(* CODESYS project amko_system.library
   Author: Chris van Kooij
   Placeholder: System_Library
   Title: System_Library
   Version: 0.0.0.3
   Description: system and module base functions
   Company: AMKO-Engineering

Project tree, tasks and I/O mapping:
  libraries: Device_Library, * (AMKO-Engineering); Tc2_Standard, * (Beckhoff Automation GmbH); Tc2_System, * (Beckhoff Automation GmbH); Tc2_Utilities, * (Beckhoff Automation GmbH); Utilities_Library, * (AMKO-Engineering)
  FaultHandler/
    function block Fb_SystemFaultHandler [ST]: CheckForModuleFaults, ExecMessageCompare, ExecScreenControl, ExecSetFaultBit, ExecWriteToLog
  GVLs/
    global variables GVL_Main
  ModuleBase/
    Base/
      function block Fb_ModuleBase [ST]: CmdAutomatic, CmdEstop, CmdHold, CmdHome, CmdInit, CmdPowerOff, CallComponents, CheckCollision, ExecAutomatic, ExecHold, ExecHome, ExecInit, ExecManual, ExecPowerOff, ExecReset, ExecSafeStop, ExecFaultHandling, ExecMainBaseFunctions
    DataTypes/
      data type Udt_ModuleBase
  SystemBase/
    DataTypes/
      data type E_StateSystem
      data type Udt_ModuleId
    program SystemBase [ST]: CallModules, ExecAutomatic, ExecHoming, ExecPowerOff, ExecSafeHold, ExecSafeReset, ExecSafeStop, Init, CallSystemFunctions, CheckSystemOK, ExecSystemRun, CmdAddModule
*)

// ModuleBase/DataTypes/Udt_ModuleBase
TYPE Udt_ModuleBase :
STRUCT
	sModuleName 		: STRING := 'NA' 		; // Module name
	bModuleActive		: 	BOOL := FALSE 		; // Module is active in the system (will be ignored by system if false) 	
	// safety Inputs
	bEstopOk			:	BOOL ; // When estop is not ok, complete machine is shut down and reinitialization is required.
	bModuleSafetyOk		: 	BOOL ; // Module safety systems are ok and safe 
	bAirPressureOk		: 	BOOL ; // system safety condition monitorring air pressure ok
	bPowerSupplyOk		: 	BOOL ; // System power supply is ok
	// main system Inputs
	bCmdStart			: 	BOOL	:= FALSE ; // System start command 
	bCmdReset 			: 	BOOL	:= FALSE ; // reset all faults 
	bCmdPowerOff		:	BOOL	:= FALSE ; // power off module 
	bCmdStartManual 	: 	BOOL 	:= FALSE ; // Start up in manual mode
 	// Com to main system
	fbFaultHandler		: 	Fb_FaultHandler 		; // Fault handler 
	sStateIndicator		: 	STRING := ''			; // Operator message, indication of current step or function 

	// Fault indications
	bMissingCond	: BOOL := FALSE ; // Module missing condition active
	bFatalFault		: BOOL := FALSE ; // Module fatal fault is active
	bCycleFault		: BOOL := FALSE ; // Module cycle fault is active

	// State indication
	bIsSafe			: BOOL := FALSE ; // Module is safe and locked until safety is ok
	bNoreference	: BOOL := FALSE ; // Module Startup Undefined initialization required

	bInitializing	: BOOL := FALSE ; // Module startup initializing
	binitialized	: BOOL := FALSE ; // Module startup initialized waiting for startup command

	bIdle 			: BOOL := FALSE ; // Module startup Idle no commands active

	bEnabling 		: BOOL := FALSE ; // Module Startup enabeling 
	bEnabled 		: BOOL := FALSE ; // Module Startup Enabled
	
	bHoming			: BOOL := FALSE ; // Module startup homing back to base position and recalibrate
	bHomed 			: BOOL := FALSE ; // Module startup homed waiting for further further commands

	bHolding 		: BOOL := FALSE ; // Module Module Hold motion command executing
	bHeld	 		: BOOL := FALSE ; // Module Hold Motion is held until command is released	
	
	bResetting 		: BOOL := FALSE ; // Module Reset resetting error status
	bResetDone 		: BOOL := FALSE ; // Module reset is done   

	bManual 		: BOOL := FALSE ; // Module Work status Module in Manual 
	bAutomatic 		: BOOL := FALSE ; // Module Work status Module in Automatic mode
	
	bPoweringOff	: BOOL := FALSE ; // Module is powering off
	bPowerdOff		: BOOL := FALSE ; // Module has powerd off 	
	
	// manual functions 
	bDevicesAddedtoManual	: BOOL := FALSE ;
	bParametersAdded		: BOOL := FALSE ;
	// Persistent data
	bCmdWritePersistent  : BOOL := false ; // write persistent data to memory
END_STRUCT
END_TYPE

// SystemBase/DataTypes/E_StateSystem
{attribute 'qualified_only'}
{attribute 'strict'}
{attribute 'to_string'}
TYPE E_StateSystem :
(
	NoReference		, 	// system has not been initialized
	Initialize		, 	// System is initializing
	LoadParameters	, 	// System is loading parameters from/to file
	Enable			, 	// System is enabling 
	Home			, 	// system is hominig 
	Reset			, 	// System is resetting
	Idle			, 	// system is waiting for commands
	Manual			, 	// System is in manual mode
	Automatic		, 	// system is in automatic mode 
	PowerOff		// system is powering off
)INT;
END_TYPE

// SystemBase/DataTypes/Udt_ModuleId
TYPE Udt_ModuleId :
STRUCT
	nNumber		: UDINT ; // Module identification number used for sorting order
	sName		: STRING; // Module name
	pFunction	: POINTER TO Fb_ModuleBase ;
END_STRUCT
END_TYPE

// GVLs/GVL_Main

{attribute 'qualified_only'} // Main system variables and state indicators
VAR_GLOBAL CONSTANT
	cnMaxNUMBEROFMODULES 	: UDINT := 10 		; // "maximum" number of modules in the system
	CtAIRPRESSUREDELAY	: TIME 	:= T#500MS	; // Timout before air fault becomes active
	cbUPSPRESENT		: BOOL	:= FALSE 	; // Enable automatic shutdown when power is interupted
END_VAR
VAR_GLOBAL PERSISTENT
	nTotalUnitsProduced		: UDINT ; // Units produced 
END_VAR

// FaultHandler/Fb_SystemFaultHandler
FUNCTION_BLOCK INTERNAL Fb_SystemFaultHandler
VAR_INPUT
	nNumberOfModules	: UDINT ; // Number of modules connected to the system fault handler
END_VAR
VAR_IN_OUT
	arpModules			: ARRAY [0..gvl_main.cnMaxNUMBEROFMODULES] OF Udt_ModuleId ;
END_VAR
VAR_OUTPUT
	// Fault types 
	bSystemFF			: BOOL 	:= FALSE	; // System fatal fault is active
	bSystemCF			: BOOL 	:= FALSE	; // System Cycle fault is active
	bSystemMC 			: BOOL 	:= FALSE	; // a missing condition is active only 
END_VAR
VAR
	// Message variables
	bResetFaults		: REFERENCE TO BOOL 	:= GVL_Message.bResetFaults		; // Reset system faults 
	bCmdSnoozeMessage	: REFERENCE TO BOOL  	:= GVL_Message.bCmdSnoozeMessage; // Snooze message display
	arActiveFaults 		: REFERENCE TO ARRAY [0..Param_Messages.nMAX_MESSAGES_SHOWN] OF UDT_Fault := GVL_Message.arActiveFaults ; // Active faults overview for showing in HMI
	arOldFaults 		: ARRAY [0..Param_Messages.nMAX_MESSAGES_SHOWN] OF UDT_Fault ; // Old faults overview for comparing to active
	arWriteToLog		: ARRAY [0..Param_Messages.nMAX_MESSAGES_SHOWN] OF UDT_Fault ; // Fault array for writing to log file 
	// Message logging
	dToday				: DATE 	; 
	nWriteStep			: UDINT := 0 ;
	bWriteError			: BOOL 	; // write to file error occured
	nWriteErroId		: UDINT ; // write error id
	// Write variables
	sActFileName		: STRING;
	hFile				: UINT	:= 0;(* File handle of the source file *)
	sMessageString		: ARRAY [0..Param_Messages.nMESSAGE_COLUMNS] OF STRING (GVL_Parameters.MAX_CSV_FIELD_LENGTH); (* temporary parameter buffer to string*)
	sCSVLine			: T_MaxString := '';(* Single CSV text line (row, record), we are using string as record buffer (your are able to see created fields) *)
	sCSVField			: T_MaxString := '';(* Single CSV field value (column, record field) *)
END_VAR
VAR // functions 
	tofSnoozeMessages	: TOF ; // timer function for message snoozing
	// Log to file functions
	fbFileOpen		: FB_FileOpen	;(* Opens file *)
	fbFileClose		: FB_FileClose	;(* Closes file *)
	fbFileGets		: FB_FileGets	;(* Reads one record (line) *)
	fbFilePuts		: FB_FilePuts	;(* Writes one record (line) *)
	fbReader		: FB_CSVMemBufferReader;(* Helper function block used to parse CSV data bytes (single record line) *)
	fbWriter		: FB_CSVMemBufferWriter;(* Helper function block used to create CSV data bytes (single record line) *)
END_VAR 
VAR CONSTANT
	stEmptyMessageUdt : UDT_Fault := (	Active 			:= FALSE,
									FaultType 		:= E_FaultTypes.NA,
									MessageNumber	:= 0,
									LocationNumber	:= 0,
									Discription 	:= '',
									LocationName	:= '',
									ComponentType	:= E_ComponentTypes.NA,
									StartTime		:= DT#2020-1-1-00:00:00,
									EndTime			:= DT#2020-1-1-00:00:00,
									FullFaultId		:= '0'	)  ;
END_VAR

// Check modules for active messages 
CheckForModuleFaults();
// set system fault bits 
ExecSetFaultBit(); 
// Message Screen controller 
ExecScreenControl();
// Log faults when they are reset
ExecMessageCompare();
// Logfile writer 
ExecWriteToLog();

METHOD PRIVATE CheckForModuleFaults : BOOL // check all modules for faults and copy them to the main fault array
VAR
	// functional variables
	i 					: UDINT ;
	j 					: UDINT ;
	// temporary fault storage
	arTempFaults	: ARRAY [0..Param_Messages.nMAX_MESSAGES_SHOWN] OF UDT_Fault ; // internal fault array
	p				: UDINT	;
END_VAR
// Go over modules to check for fault messages 
FOR i := 0 TO nNumberOfModules DO 
	// Check for active messages
	FOR j := 0 TO Param_Messages.nMAX_MESSAGES_SHOWN DO 
		IF arpModules[i].pFunction^.fbFaultHandler.arActiveFaults[j].FaultType <> E_FaultTypes.NA THEN 
			arTempFaults[p]:= arpModules[i].pFunction^.fbFaultHandler.arActiveFaults[j] ;
			p := MAX( p + 1, Param_Messages.nMAX_MESSAGES_SHOWN)  ;
		ELSE
			EXIT ;
		END_IF
	END_FOR
END_FOR

arOldFaults		:= arActiveFaults 	;
arActiveFaults	:= arTempFaults 	;
END_METHOD

METHOD PRIVATE ExecMessageCompare : BOOL
VAR
	// functional variables
	i 			: UDINT ;
	j 			: UDINT ;
	bFaultFound : BOOL ;
	p			: UDINT;
END_VAR
// Check if any changes occured in the active faults
FOR i := 0 TO Param_Messages.nMAX_MESSAGES_SHOWN DO
	// break loop if fault is empty
	IF  arOldFaults[i].FaultType = E_FaultTypes.NA THEN  
		EXIT;
	ELSE
		// check if the fault is still active
		bFaultFound := TRUE; 
		FOR j := 0 TO Utilities_Library.Param_Messages.nMAX_MESSAGES_SHOWN DO
			bFaultFound := arOldFaults[i].FullFaultId = arActiveFaults[j].FullFaultId AND bFaultFound ;
		END_FOR
		// if the fault is not faund then wrtie it to the logging array for loging
		IF NOT bFaultFound THEN 
			arWriteToLog[p] := arOldFaults[i] ;
			p := p + 1 ; 
		END_IF
	END_IF
END_FOR
END_METHOD

METHOD PRIVATE ExecScreenControl : BOOL // Control message screen 
VAR_INPUT
END_VAR
tofSnoozeMessages(IN := bCmdSnoozeMessage, PT := GVL_Message.tMESSAGESNOOZEDURATION);

// Set screen control 
IF bSystemCF OR bSystemFF THEN 
	GVL_Message.bHideFaults := FALSE ;
ELSIF bSystemMC AND NOT tofSnoozeMessages.Q THEN 
	GVL_Message.bHideFaults := FALSE ;
ELSE
	GVL_Message.bHideFaults := TRUE ;
END_IF
END_METHOD

METHOD PRIVATE ExecSetFaultBit : BOOL
VAR
	// functional variables
	i 			: UDINT ;
END_VAR
bSystemFF	:= FALSE ;
bSystemCF	:= FALSE ;
bSystemMC	:= FALSE ;

FOR i := 0 TO Param_Messages.nMAX_MESSAGES_SHOWN DO
	bSystemFF	:= arActiveFaults[i].FaultType = E_FaultTypes.FF OR bSystemFF;
	bSystemCF	:= arActiveFaults[i].FaultType = E_FaultTypes.CF OR bSystemCF;
	bSystemMC	:= arActiveFaults[i].FaultType = E_FaultTypes.MC OR bSystemMC;
END_FOR
END_METHOD

METHOD PRIVATE ExecWriteToLog : BOOL
VAR 
	i : UDINT ; 
	p : UDINT ; // Fault array pointer
END_VAR
dToday := DT_TO_DATE(Sys_Variables.SystemTime);
// create file name with Current date 
sActFileName 	:= CONCAT(STR1 := Param_Messages.sLOGFILE_PATH	, STR2 := Param_Messages.sLOGFILE_NAME	);
sActFileName 	:= CONCAT(STR1 := sActFileName					, STR2 := DATE_TO_STRING(dToday)		);
sActFileName 	:= CONCAT(STR1 := sActFileName					, STR2 := '.csv'						);

// ===== Start file write =====
CASE nWriteStep OF
	0:	(* Wait until log array is filled *)
		IF arWriteToLog[0].FaultType <> E_FaultTypes.NA THEN 
			hFile				:= 0;
			nWriteStep 			:= 1;
		ELSE 
			RETURN ;
		END_IF
	1:	(* Open source file *)
		fbFileOpen(  bExecute := FALSE  );
		fbFileOpen( sNetId := GVL_Parameters.sNetId, sPathName := sActFileName , nMode := FOPEN_MODEAPPEND OR FOPEN_MODETEXT,(* Open file in TEXT mode! *)
					ePath := PATH_GENERIC, bExecute := TRUE );
		nWriteStep := nWriteStep + 1 ;
	2:(* Wait until open not busy *)
		fbFileOpen( bExecute := FALSE, bError => bWriteError, nErrID => nWriteErroId, hFile => hFile );
		IF NOT fbFileOpen.bBusy THEN
			IF NOT fbFileOpen.bError THEN
				nWriteStep := nWriteStep + 1 ;
			ELSE(* Error: file not found? *)
				nWriteStep := 100;
			END_IF
		END_IF
	3: (* Check if faultrecord is active if so skip record *)
		nWriteStep := nWriteStep + 1 ;
	4:(* Convert one PLC record to CSV format *)
		sCSVLine := '';
		fbWriter.eCmd := eEnumCmd_First;(* Write first field value *)
		// write message data to string
		sMessageString[0] 	:= TO_STRING(arWriteToLog[p].FaultType				);
		sMessageString[1]	:= DT_TO_STRING(arWriteToLog[p].StartTime			);
		sMessageString[2]	:= DT_TO_STRING(Sys_Variables.SystemTime			);
		sMessageString[3]	:= UDINT_TO_STRING(arWriteToLog[p].MessageNumber	);
		sMessageString[4]	:= UDINT_TO_STRING(arWriteToLog[p].LocationNumber	); 
		sMessageString[5]	:= arWriteToLog[p].Discription						;
		sMessageString[6]	:= arWriteToLog[p].LocationName						;
		sMessageString[7]	:= TO_STRING(arWriteToLog[p].ComponentType			);
		// write data to .csv buffer 
		FOR i := 0 TO Param_Messages.nMESSAGE_COLUMNS BY 1 DO
			sCSVField := STRING_TO_CSVFIELD(in :=  sMessageString[i], FALSE );
			(* Add new field to the record buffer *)
			fbWriter( 	pBuffer := ADR( sCSVLine ), cbBuffer := SIZEOF( sCSVLine ) - 1, putValue := sCSVField, pValue := 0, cbValue := 0,
						bCRLF := ( i = Param_Messages.nMESSAGE_COLUMNS ) );(* bCRLF == TRUE => Write CRLF after the last field value *)
			IF fbWriter.bOk THEN
				fbWriter.eCmd := eEnumCmd_Next;
			ELSE
				nWriteStep := 100;
				RETURN;
			END_IF
		END_FOR(* FOR nColumn := 0... *)

		(* FB_FilePuts adds allready CR (carriage return) to the written line.
		We have to replace the $R$L characters with $L character to avoid double CR. *)
		IF RIGHT( sCSVLine, 2 ) = '$R$L' THEN
			sCSVLine := REPLACE( sCSVLine, '$L', 2, LEN( sCSVLine ) - 1 );
		END_IF
		nWriteStep := nWriteStep + 1 ;
	5:	(* Write single text line to file *)
		fbFilePuts( bExecute := FALSE );
		fbFilePuts( sNetId := GVL_Parameters.sNetId, hFile := hFile, sLine := sCSVLine, bExecute := TRUE );
		nWriteStep := nWriteStep + 1 ;
	6:(* Wait until write not busy *)
		fbFilePuts( bExecute := FALSE, bError => bWriteError, nErrID => nWriteErroId );
		IF NOT fbFilePuts.bBusy THEN
			IF NOT fbFilePuts.bError THEN
				nWriteStep := nWriteStep + 1 ;
			ELSE(* Error *)
				nWriteStep := 100;
			END_IF
		END_IF
	7: (* clear fault from array and go to next fault *)
		arWriteToLog[p]:= stEmptyMessageUdt;
		IF p < Param_Messages.nMAX_MESSAGES_SHOWN THEN 
			p := p +1 ;
		END_IF
		nWriteStep := nWriteStep +1 ;
	8: (* If fault is active then repeat previous step, else close file*)		
		IF  arWriteToLog[p].FaultType <> E_FaultTypes.NA THEN 
			nWriteStep := 3 ;
		ELSE
			nWriteStep := 10;
		END_IF
	10:	(* Close source file *)
		fbFileClose( bExecute := FALSE );
		fbFileClose( sNetId := GVL_Parameters.sNetId, hFile := hFile, bExecute := TRUE );
		nWriteStep := 11;
	11:(* Wait until close not busy *)
		fbFileClose( bExecute := FALSE, bError => bWriteError, nErrID => nWriteErroId );
		IF ( NOT fbFileClose.bBusy ) THEN
			hFile 		:= 0;
			nWriteStep 	:= 100;
		END_IF
	100: (* Error or ready nWriteStep => cleanup *)
		IF ( hFile <> 0 ) THEN
			nWriteStep	:= 10; (* Close the source file *)
		ELSE
			nWriteStep 	:= 0;	(* Ready *)
			ExecWriteToLog := TRUE ;
		END_IF
END_CASE
END_METHOD

END_FUNCTION_BLOCK

// ModuleBase/Base/Fb_ModuleBase
{attribute 'reflection'}
FUNCTION_BLOCK PUBLIC ABSTRACT Fb_ModuleBase
VAR_INPUT
	nModuleID			: 	UDINT 	:= 1 	; // module reference number used for fault, enable, reset, and safety functions (default := 1, 0 = main system)
	// main system Inputs
	bEnable				: 	BOOL	:= FALSE ; // (autolinked) module enable 	
	bCmdReset 			: 	BOOL	:= FALSE ; // (AutoLinked) reset all faults 
	bSysFatalFault		: 	BOOL 	:= FALSE ; // (AutoLinked) System fatal fault active
	bSysCycleFault		: 	BOOL 	:= FALSE ; // (AutoLinked) System fatal fault active 
	// Internal safety 
	bSafetyOK			: BOOL := FALSE ; // Module internal safety is ok
END_VAR
VAR_OUTPUT
	sName 				: STRING 	:= 'NA' 			; // Module name
	bAddedToSystem		: BOOL 		:= FALSE 			; // module has been added to the system
 	// Com to main system
	fbFaultHandler		: 	Fb_FaultHandler 		; // Fault handler 
	sStateIndicator		: 	STRING := ''			; // Operator message, indication of current step or function 

	// Fault indications
	bMissingCond	: BOOL := FALSE ; // Module missing condition active
	bFatalFault		: BOOL := FALSE ; // Module fatal fault is active
	bCycleFault		: BOOL := FALSE ; // Module cycle fault is active

	// State indication
	bIsSafe			: BOOL := FALSE ; // Module is safe and locked until safety is ok
	bNoreference	: BOOL := FALSE ; // Module Startup Undefined initialization required
	binitialized	: BOOL := FALSE ; // Module startup initialized waiting for startup command
	bHomed 			: BOOL := FALSE ; // Module startup homed waiting for further further commands

	bHolding 		: BOOL := FALSE ; // Module Module Hold motion command executing
	bHeld	 		: BOOL := FALSE ; // Module Hold Motion is held until command is released	
	
	bResetDone 		: BOOL := FALSE ; // Module reset is done   

	bManual 		: BOOL := FALSE ; // Module Work status Module in Manual
	bStartAuto		: BOOL := FALSE ; // Module start automatic cycle 
	bAutomatic 		: BOOL := FALSE ; // Module Work status Module in Automatic mode
	
	bPoweringOff	: BOOL := FALSE ; // Module is powering off
	bPowerdOff		: BOOL := FALSE ; // Module has powerd off 	

END_VAR
VAR 
	// manual functions 
	bParametersAdded		: BOOL := FALSE ;
	// Persistent data
	bCmdWritePersistent  : BOOL := false ; // write persistent data to memory
	// Module data
	stMessage				: UDT_Fault			; // Message data
	// Function path 
	{attribute 'instance-path'} 
    {attribute 'noinit'}
	sPath			: STRING	; // Path name of function (used for manual reference)
END_VAR


// Get device name from function
IF sName = 'NA' THEN 
	sName := F_FBNameFromPath(sPath := sPath);
END_IF

// Add module to system
IF NOT bAddedToSystem THEN
	bAddedToSystem S= SystemBase.CmdAddModule(refToModule := THIS^);
END_IF

// Execute functions
ExecMainBaseFunctions();

METHOD INTERNAL CmdAutomatic : BOOL
VAR_INPUT
END_VAR
bStartAuto 		:= TRUE ;

CmdAutomatic 	:= bAutomatic;
END_METHOD

METHOD INTERNAL CmdEstop : BOOL
VAR_INPUT
END_VAR
ExecSafeStop();
bHomed			:= FALSE ;
bAutomatic 		:= FALSE ;


CmdEstop := bIsSafe ;
END_METHOD

METHOD INTERNAL CmdHold : BOOL
VAR_INPUT
END_VAR
bAutomatic 	:= FALSE ;
ExecHold();


CmdHold := bHeld ;
END_METHOD

METHOD INTERNAL CmdHome : BOOL
VAR_INPUT
END_VAR
ExecHome();

CmdHome := bHomed;
END_METHOD

METHOD INTERNAL CmdInit : BOOL
VAR_INPUT
END_VAR
ExecInit();

CmdInit := binitialized;
END_METHOD

METHOD INTERNAL CmdPowerOff : BOOL
VAR_INPUT
END_VAR
ExecPowerOff();
bAutomatic := FALSE ;

CmdPowerOff := bPowerdOff;
END_METHOD

METHOD PROTECTED ABSTRACT CallComponents : BOOL
VAR_INPUT
END_VAR
END_METHOD

METHOD PUBLIC ABSTRACT CheckCollision : BOOL // Checks device commands for positble collisions  and block if necesarry
VAR_INPUT
END_VAR
END_METHOD

METHOD PROTECTED ABSTRACT ExecAutomatic : BOOL
VAR_INPUT
END_VAR
END_METHOD

METHOD PROTECTED ABSTRACT ExecHold : BOOL
VAR_INPUT
END_VAR
END_METHOD

METHOD PROTECTED ABSTRACT ExecHome : BOOL
VAR_INPUT
END_VAR
END_METHOD

METHOD PROTECTED ABSTRACT ExecInit : BOOL
VAR_INPUT
END_VAR
END_METHOD

METHOD PROTECTED ExecManual : BOOL
VAR_INPUT
END_VAR
END_METHOD

METHOD PROTECTED ABSTRACT ExecPowerOff : BOOL
VAR_INPUT
END_VAR
END_METHOD

METHOD PROTECTED ABSTRACT ExecReset : BOOL
VAR_INPUT
END_VAR
END_METHOD

METHOD PROTECTED ABSTRACT ExecSafeStop : BOOL
VAR_INPUT
END_VAR
END_METHOD

METHOD ExecFaultHandling : BOOL
VAR_INPUT
END_VAR
// Call reset functions
IF bCmdReset THEN 
	fbFaultHandler.bReset := TRUE ;
	ExecReset();
END_IF

// Call message function
fbFaultHandler(bReset := bCmdReset);

bFatalFault := fbFaultHandler.bActFF ;
bCycleFault := fbFaultHandler.bActCF ;

IF bFatalFault THEN
	ExecSafeStop()	;
	binitialized	:= FALSE; 
	bHomed			:= FALSE;
ELSIF bCycleFault THEN
	bHeld			S= ExecHold();
	bHolding 		:= NOT bHeld ;
END_IF

// Reset safe state when enable is active
bIsSafe R= bEnable ;

// Prevent automatic start when fault is active
bStartAuto R= bCmdReset OR bFatalFault OR bCycleFault ;
END_METHOD

METHOD INTERNAL ExecMainBaseFunctions : BOOL
VAR_INPUT
END_VAR
// Check for anny Internal collisions
CheckCollision();

// Call components 
CallComponents();

// Call fault handling function 
ExecFaultHandling();

// Run automatic function 
IF bStartAuto THEN 
	bAutomatic := ExecAutomatic();
	bStartAuto :=FALSE ;
ELSE
	bAutomatic := FALSE ;
END_IF

// Persistent data 
IF bCmdWritePersistent THEN 
	bCmdWritePersistent R= DataManager.FbPersistentManager.Write();
END_IF
END_METHOD

END_FUNCTION_BLOCK

// SystemBase/SystemBase
{attribute 'reflection'}
PROGRAM SystemBase // system base program, from here all modules are controlled and the system functions are called.
VAR_IN_OUT
	// HMI Screens 
	nHMIShownscreen	: INT ; // show visualization screen (0 = default home screen, 1 = automatic screen, 2 =< configurable) 
END_VAR
VAR
	// Fault indications
	bMissingCond	: BOOL := FALSE ; // Module missing condition active
	bFatalFault		: BOOL := FALSE ; // Module fatal fault is active
	bCycleFault		: BOOL := FALSE ; // Module cycle fault is active

	// State indication
	bIsSafe			: BOOL := FALSE ; // Module is safe and locked until safety is ok
	bNoreference	: BOOL := FALSE ; // Module Startup Undefined initialization required

	bInitializing	: BOOL := FALSE ; // Module startup initializing
	binitialized	: BOOL := FALSE ; // Module startup initialized waiting for startup command

	bIdle 			: BOOL := FALSE ; // Module startup Idle no commands active

	bEnabling 		: BOOL := FALSE ; // Module Startup enabeling 
	bEnabled 		: BOOL := FALSE ; // Module Startup Enabled
	
	bHoming			: BOOL := FALSE ; // Module startup homing back to base position and recalibrate
	bHomed 			: BOOL := FALSE ; // Module startup homed waiting for further further commands

	bHolding 		: BOOL := FALSE ; // Module Module Hold motion command executing
	bHeld	 		: BOOL := FALSE ; // Module Hold Motion is held until command is released	
	
	bResetting 		: BOOL := FALSE ; // Module Reset resetting error status
	bResetDone 		: BOOL := FALSE ; // Module reset is done   

	bManual 		: BOOL := FALSE ; // Module Work status Module in Manual 
	
	bStartAuto		: BOOL := FALSE ; // Start automatic mode
	bAutomatic 		: BOOL := FALSE ; // Module Work status Module in Automatic mode
	
	bPoweringOff	: BOOL := FALSE ; // Module is powering off
	bPowerdOff		: BOOL := FALSE ; // Module has powerd off 	

END_VAR
VAR
	// System inputs 
	ibEstopOk 			AT%I*	: BOOL  ; // system emergency stop ok
	ibSystemSafetyOK	AT%I*	: BOOL  ; // System is safe 
	ibPowerSupplyOk	 	AT%I*	: BOOL  ; // System Power supply is ok 
	fbAirpressureOk 			: Fb_DevDigitalInputFunctions  	; // system airpressure is ok
	fbCmdResetSafety		 	: FB_DevPushbuttonLight 		; // System reset
	
	// System safety valve
	fbValveMainAirSupply		: FB_DevValve ; // Main air supply valve 
	
	// system Commands 
	fbCmdStartSystem		 	: FB_DevPushbuttonLight  		; // (re)start system input from button
	fbCmdStartManual			: FB_DevHMIButton 				; // Start system in manual mode 
	fbCmdPowerOff				: FB_DevHMIButton 				; // Power off system
	
	//System state
	bSystemOK				: BOOL := FALSE ; // all safety and vitals are OK
	eStateSystem			: E_StateSystem := E_StateSystem.NoReference ; // State of system

	// Set system variables
	fbSetSystemVariables	: Fb_SystemVariables ;
	
	// System Fault handling
	fbSystemFaultHandler	: Fb_SystemFaultHandler ;
	fbOperatorMessage		: FB_OperatorMessageDisplay ; //Operator message or system state message hadler 
	
 	// Module states
	nNumberOfModules	: UDINT := 0 ; // Number of modules added to the system 
	arpModules			: ARRAY [0..gvl_main.cnMaxNUMBEROFMODULES] OF Udt_ModuleId ; 

	// power down system function
	ntShutDown			: NT_Shutdown ; // shutdown system function 

	// Manual controller
	bDevicesAddedtoManual : BOOL := FALSE ; // Add system device (buttons) to manual controller

	// Function path 
	{attribute 'instance-path'} 
    {attribute 'noinit'}
	sPath			: STRING	; // Path name of function (used for manual reference
END_VAR

// check if at least one module is added else return 
IF arpModules[0].pFunction = 0 THEN 
	RETURN;
END_IF

// check functions
CheckSystemOK();

// Run system
ExecSystemRun();

// call device functions 
CallSystemFunctions();

// Call modules 
CallModules();

METHOD PRIVATE CallModules : BOOL
VAR
	i : UDINT ;
END_VAR
// set base conditions
bIsSafe		:= TRUE ;
bIdle		:= TRUE ;	
bHeld		:= TRUE ;
bResetDone 	:= TRUE	;
bManual		:= TRUE	;
bAutomatic	:= TRUE	;
bEnabled	S= bEnabling ;

// copy inputs to modules 
FOR i := 0 TO nNumberOfModules DO 
	// set system commands
	arpModules[i].pFunction^.bEnable			:= bEnabled		;
	arpModules[i].pFunction^.bCmdReset			:= bResetting	;
	arpModules[i].pFunction^.bSafetyOK			:= bSystemOK	;
	// Read state indications 
	bIsSafe 	:= arpModules[i].pFunction^.bIsSafe AND bIsSafe ;
	bEnabled 	:= arpModules[i].pFunction^.bEnable AND bEnabled  ;
	bEnabling	R= bEnabled ;
	bHeld		:= arpModules[i].pFunction^.bHeld AND bHeld ;
	bHolding	R= bHeld ;
	bResetDone	:= arpModules[i].pFunction^.bResetDone AND bResetDone ;
	bResetting	R= bResetDone ;
	bManual		:= arpModules[i].pFunction^.bManual AND bManual ;
	bAutomatic	:= arpModules[i].pFunction^.bAutomatic AND bAutomatic ;
	bStartAuto	R= bAutomatic ;
END_FOR
END_METHOD

METHOD PRIVATE ExecAutomatic : BOOL
VAR_INPUT
END_VAR
VAR
	i : UDINT ;
END_VAR
// Run automatic function in 
FOR i := 0 TO nNumberOfModules DO 
	arpModules[i].pFunction^.CmdAutomatic() ;
END_FOR

// Set Start button state
IF bAutomatic THEN 
	fbCmdStartSystem.CmdOn();
ELSE
	fbCmdStartSystem.CmdBlinkFast();
END_IF

ExecAutomatic := bAutomatic;
END_METHOD

METHOD PRIVATE ExecHoming : BOOL
VAR_INPUT
END_VAR
VAR
	i : UDINT ;
END_VAR
// Home all modules
bHomed	:= TRUE;
FOR i := 0 TO nNumberOfModules DO 
	IF NOT arpModules[i].pFunction^.bHomed THEN 
		arpModules[i].pFunction^.CmdHome();
	END_IF
	bHomed 	:= bHomed AND arpModules[i].pFunction^.bHomed;
	bHoming	:= NOT bHomed ;
 END_FOR
 
 ExecHoming := bHomed ;
END_METHOD

METHOD PRIVATE ExecPowerOff : BOOL
VAR_INPUT
END_VAR
VAR 
	i : UDINT ;
END_VAR
// Power off all modules
bPowerdOff	:= TRUE;
FOR i := 0 TO nNumberOfModules DO 
	bPowerdOff 		:= arpModules[i].pFunction^.CmdPowerOff () AND bPowerdOff ;
	bPoweringOff	:= NOT bPowerdOff ;
 END_FOR
 
 ExecPowerOff := bPowerdOff ;
END_METHOD

METHOD PRIVATE ExecSafeHold : BOOL
VAR_INPUT
END_VAR
VAR
	i : UDINT ;
END_VAR
// Hold all modules
bEnabled		:= FALSE;
bEnabling		:= FALSE;
bHoming			:= FALSE;
bStartAuto		:= FALSE;

bHeld	:= TRUE;
FOR i := 0 TO nNumberOfModules DO 
	bHeld	:= bHeld AND	arpModules[i].pFunction^.CmdHold();
	bHolding:= NOT bHeld ;
END_FOR
 
 ExecSafeHold := bHeld ;
END_METHOD

METHOD PRIVATE ExecSafeReset : BOOL
VAR_INPUT
END_VAR
END_METHOD

METHOD PRIVATE ExecSafeStop : BOOL
VAR_INPUT
END_VAR
VAR
	i : UDINT ;
END_VAR
// perform Estop for all modules
bEnabled		:= FALSE;
bEnabling		:= FALSE;
bInitializing	:= FALSE;
bHoming			:= FALSE;
bStartAuto		:= FALSE;

// Close and vent main air supply
fbValveMainAirSupply.CmdClose();

// Module safe stop
bIsSafe			:= TRUE	;
FOR i := 0 TO nNumberOfModules DO 
	bIsSafe	:= bIsSafe AND	arpModules[i].pFunction^.CmdEstop();
END_FOR

IF bIsSafe THEN 
	fbValveMainAirSupply.CmdSafeStop();
END_IF
 
ExecSafeStop := bIsSafe ;
END_METHOD

METHOD PRIVATE Init : BOOL
VAR_INPUT
END_VAR
VAR
	i : UDINT ;
END_VAR
// initialize system functions
fbValveMainAirSupply.Init(	nDevNumber 	:= 1,
							eResetState	:= E_ValveResetState.Res_Closed,
							eSafeState	:= E_ValveResetState.Res_Closed);


							
// Initialize all modules
binitialized	:= TRUE ;
FOR i := 0 TO nNumberOfModules DO 
	IF NOT arpModules[i].pFunction^.binitialized THEN 
		arpModules[i].pFunction^.CmdInit();
	END_IF
	binitialized 	:= binitialized AND arpModules[i].pFunction^.binitialized;
	bInitializing 	:= NOT binitialized ;
	// Set feedback to screen (needs to be added)
 END_FOR
 
 Init := binitialized ;
END_METHOD

METHOD PRIVATE CallSystemFunctions : BOOL
VAR_INPUT
END_VAR
// set system variables 
fbSetSystemVariables();

// call parameter handler
GVL_Parameters.fbParameterHandler();
GVL_DevManual.fbManualControler();

// Execute button functions 
fbCmdStartSystem();
fbCmdResetSafety(); 
// execute input functions
fbAirpressureOk();
fbValveMainAirSupply(	nModuleId	:= 0,
						bEnable		:= TRUE,
						bSafetyOk	:= ibEstopOk,
						bReset		:= GVL_Message.bResetFaults);
// Call persistent data handler 
DataManager.FbPersistentManager();

// Add device functions to manual controller 
IF NOT bDevicesAddedtoManual THEN
	GVL_DevManual.fbManualControler.CmdAddDevice( refToDevice := fbAirpressureOk 	);
	GVL_DevManual.fbManualControler.CmdAddDevice( refToDevice := fbCmdStartSystem	);
	GVL_DevManual.fbManualControler.CmdAddDevice( refToDevice := fbCmdResetSafety	);
	bDevicesAddedtoManual S= TRUE ;
END_IF
END_METHOD

METHOD PRIVATE CheckSystemOK : BOOL
VAR
	i : UDINT ;
END_VAR
// shutdown emediately if power is down 
ntShutDown(START := bPowerdOff OR (NOT ibPowerSupplyOk AND GVL_Main.cbUPSPRESENT));

// Call faulthandler
fbSystemFaultHandler( 	nNumberOfModules	:= nNumberOfModules,
						arpModules			:= arpModules,
						bSystemFF			=> bFatalFault,
						bSystemCF			=> bCycleFault,
						bSystemMC			=> bMissingCond);

// Check system safety and Faults
IF NOT ibEstopOk OR NOT ibPowerSupplyOk OR bFatalFault THEN 
	ExecSafeStop();
ELSIF NOT ibSystemSafetyOK OR NOT fbAirpressureOk.bFcoDelay OR bCycleFault  THEN
	ExecSafeHold();
ELSIF (bIsSafe OR bHeld)  THEN 
	bSystemOK S= TRUE ;	
END_IF

bSystemOK R= NOT (ibEstopOk AND ibPowerSupplyOk AND ibSystemSafetyOK AND fbAirpressureOk.bFcoDelay);

// Set safety state and button light state
fbCmdResetSafety.bEnable S= TRUE ;
IF NOT ibEstopOk THEN 
	fbCmdResetSafety.CmdOn() ;
ELSIF NOT ibSystemSafetyOK THEN 
	fbCmdResetSafety.CmdBlinkSlow() ;
ELSIF NOT fbAirpressureOk.bFcoDelay THEN
	fbCmdResetSafety.CmdBlinkFast() ;
END_IF

// Main air control 
IF ibEstopOk AND 
	ibSystemSafetyOK AND 
	ibPowerSupplyOk AND
	binitialized AND 
	NOT bFatalFault THEN 
fbValveMainAirSupply.CmdOpen();
END_IF
END_METHOD

METHOD INTERNAL ExecSystemRun : BOOL
VAR_INPUT
END_VAR
// set system variables 
fbSetSystemVariables();

// Check for system commands
IF eStateSystem > E_StateSystem.Enable THEN 
	IF GVL_Message.bResetFaults OR fbCmdResetSafety.bFeStatus THEN
		bResetDone		:= FALSE ;
		eStateSystem 	:= E_StateSystem.Reset ;
	ELSIF fbCmdResetSafety.bFcoDelay THEN 
		eStateSystem := E_StateSystem.NoReference ;
	ELSIF fbCmdPowerOff.bFcoDelay THEN 
		eStateSystem := E_StateSystem.PowerOff ;
	ELSIF bFatalFault THEN 
		eStateSystem := E_StateSystem.Enable;
	ELSIF bCycleFault THEN 
		IF eStateSystem > E_StateSystem.Idle THEN
			eStateSystem := E_StateSystem.Idle ;
		ELSE
			eStateSystem := E_StateSystem.Enable ;
		END_IF
	ELSIF fbCmdStartSystem.bFeStatus THEN 
		bStartAuto := TRUE ;
	END_IF
	
// Check for safety state
	IF NOT ibEstopOk OR NOT fbAirpressureOk.bFcoDelay THEN
		eStateSystem := E_StateSystem.Enable ;
	ELSIF NOT ibSystemSafetyOK THEN
		IF eStateSystem > E_StateSystem.Idle THEN
			eStateSystem := E_StateSystem.Idle ;
		ELSE
			eStateSystem := E_StateSystem.Enable ;
		END_IF
	END_IF
ELSE 
	IF GVL_Message.bResetFaults OR fbCmdResetSafety.bFeStatus THEN
		bResetDone := FALSE ;
		bResetting := TRUE ;
	END_IF
END_IF

// add manual function	
	
// State machine 
CASE eStateSystem OF 
	E_StateSystem.NoReference:
		nHMIShownscreen := 0 ;
		binitialized 	:= FALSE ;
		bHomed			:= FALSE ;
		bEnabled		:= FALSE ;
		IF bIsSafe THEN 
			eStateSystem := E_StateSystem.Initialize ;
		END_IF
	E_StateSystem.Initialize:
		IF Init() THEN
			eStateSystem := E_StateSystem.LoadParameters	;
		END_IF
	E_StateSystem.LoadParameters:
		IF GVL_Parameters.fbParameterHandler.Init() THEN
			eStateSystem := E_StateSystem.Enable ;
		END_IF
	E_StateSystem.Enable:
		nHMIShownscreen := 0 ;
		IF bEnabled THEN 
			eStateSystem := E_StateSystem.Home ;
		ELSIF GVL_DevManual.bManualModeActive THEN
			eStateSystem := E_StateSystem.Manual ;
		ELSE
			bEnabling 	:= bSystemOK;
		END_IF
	E_StateSystem.Home:
		IF ExecHoming() THEN
			eStateSystem := E_StateSystem.Idle;
		END_IF
	E_StateSystem.Reset:
		nHMIShownscreen := 0 ;
		IF bResetDone AND bHomed THEN
			eStateSystem := E_StateSystem.Idle ;
		ELSIF bResetDone THEN 
			eStateSystem := E_StateSystem.Enable ;
		ELSE
			bResetting S= TRUE ;
		END_IF
	E_StateSystem.Idle:
		nHMIShownscreen := 0 ;
		IF bSystemOK AND NOT bHeld AND bStartAuto THEN
			nHMIShownscreen := 1 ;
			eStateSystem := E_StateSystem.Automatic ;
		ELSIF bSystemOK AND GVL_DevManual.bManualModeActive THEN
			eStateSystem	:= E_StateSystem.Manual ;
		END_IF
	E_StateSystem.Automatic:
			ExecAutomatic();
			IF bAutomatic AND fbCmdStartSystem.bFeStatus THEN 
				eStateSystem := E_StateSystem.Idle ;
			END_IF
	E_StateSystem.Manual:
			IF NOT GVL_DevManual.bManualModeActive THEN 
				eStateSystem := E_StateSystem.Enable ;
			END_IF
	E_StateSystem.PowerOff:
		ExecPowerOff();
	ELSE 
		;		
END_CASE
END_METHOD

METHOD PUBLIC CmdAddModule : BOOL
VAR_INPUT
	refToModule : REFERENCE TO Fb_ModuleBase ; // reference to module function
END_VAR
VAR
	bModuleAdded	: BOOL ;
	i 				: UDINT ; 
END_VAR
// Check if device is not already in the array 
FOR i:= 0 TO GVL_Main.cnMaxNUMBEROFMODULES DO
	IF arpModules[i].pFunction = 0 THEN 
		nNumberOfModules:= i;
		EXIT;	
	ELSIF arpModules[i].sName = refToModule.sName THEN 
		bModuleAdded := TRUE ;
	ELSE
		RETURN;
	END_IF 
END_FOR

// If device is not found add device to the list
IF NOT bModuleAdded THEN 
	nNumberOfModules := LIMIT(0, nNumberOfModules,GVL_Main.cnMaxNUMBEROFMODULES)	;
	arpModules[nNumberOfModules].nNumber 	:= refToModule.nModuleID;
	arpModules[nNumberOfModules].sName		:= refToModule.sName	;
	arpModules[nNumberOfModules].pFunction 	:= ADR(refToModule)		;	
	bModuleAdded := TRUE ;
END_IF

CmdAddModule := bModuleAdded ;
END_METHOD

END_PROGRAM
